{attribute 'qualified_only'}
{attribute 'strict'}
{attribute 'to_string'}
TYPE EN_TrayFeederMessaging :
(
	waitInitStart			:=0,
	initFinished			:=999,
	
	autoStart				:=1000,
	readyToScan				:=1400,
	scanning				:=1410,
	scanFinished			:=1490,
	readyToPick				:=1500,
	picking					:=1510,
	pickFinished			:=1590,
	autoProcessFinished		:=1999
)DINT := waitInitStart;
END_TYPE

(* stored: Version 1.1.0.1, ProductVersion 3.1.4024.12
   DUT EN_TrayFeederMessaging: Id {0f8b0073-a2d8-463c-968c-eb611f66abb7} *)
